INTERFACE IF_Actuator
	//// Generic Interface for actuators

METHOD Disable : BOOL
VAR_INPUT
END_VAR
END_METHOD

METHOD Enable : BOOL
VAR_INPUT
END_VAR
END_METHOD

METHOD GetStatus : ST_ActuatorStatus
VAR_INPUT
END_VAR
END_METHOD

METHOD Reset : BOOL
VAR_INPUT
END_VAR
END_METHOD

END_INTERFACE

(* stored: Version 1.1.0.1, ProductVersion 3.1.4024.12
   Itf IF_Actuator: Id {7b6b94f4-376b-4427-aad2-3ea78a291535}
   Method Disable: Id {220ecdfe-9298-4831-b70c-4ff1ae259ea8}
   Method Enable: Id {527926bf-2005-44c2-b59f-9b58d7af006a}
   Method GetStatus: Id {3a0ea259-0c66-4849-a9ae-118b565beaf2}
   Method Reset: Id {661b6735-cc7f-406b-9834-be016524e121} *)
